TYPE ST_ToolData :
STRUCT
END_STRUCT
END_TYPE

(* stored: Version 1.1.0.1, ProductVersion 3.1.4022.18
   DUT ST_ToolData: Id {786298c7-d114-49c2-90d8-c0defcc60f2f} *)
